DATA_BLOCK "INST_GN BLOKADA_SRUBY_LEWY"
{ S7_Optimized_Access := 'TRUE' }
VERSION : 0.1
NON_RETAIN
"3STATE_PISTON_with_brake"

BEGIN

END_DATA_BLOCK

DATA_BLOCK "INST_GN BLOKADA_SRUBY_SRODEK"
{ S7_Optimized_Access := 'TRUE' }
VERSION : 0.1
NON_RETAIN
"3STATE_PISTON_with_brake"

BEGIN

END_DATA_BLOCK

DATA_BLOCK "INST_GN BLOKADA_SRUBY_PRAWY"
{ S7_Optimized_Access := 'TRUE' }
VERSION : 0.1
NON_RETAIN
"3STATE_PISTON_with_brake"

BEGIN

END_DATA_BLOCK

DATA_BLOCK "INST_GN ZASUWKA"
{ S7_Optimized_Access := 'TRUE' }
VERSION : 0.1
NON_RETAIN
"3STATE_PISTON_with_brake"

BEGIN

END_DATA_BLOCK

DATA_BLOCK "INST_BR PIN_PODNOSZENIE_01"
{ S7_Optimized_Access := 'TRUE' }
VERSION : 0.1
NON_RETAIN
"3STATE_PISTON_with_brake"

BEGIN

END_DATA_BLOCK

DATA_BLOCK "INST_BR PIN_01"
{ S7_Optimized_Access := 'TRUE' }
VERSION : 0.1
NON_RETAIN
"3STATE_PISTON_with_brake"

BEGIN

END_DATA_BLOCK

DATA_BLOCK "INST_BR PIN_PODNOSZENIE_02"
{ S7_Optimized_Access := 'TRUE' }
VERSION : 0.1
NON_RETAIN
"3STATE_PISTON_with_brake"

BEGIN

END_DATA_BLOCK

DATA_BLOCK "INST_BR PIN_02"
{ S7_Optimized_Access := 'TRUE' }
VERSION : 0.1
NON_RETAIN
"3STATE_PISTON_with_brake"

BEGIN

END_DATA_BLOCK

DATA_BLOCK "INST_BR PIN_PODNOSZENIE_03"
{ S7_Optimized_Access := 'TRUE' }
VERSION : 0.1
NON_RETAIN
"3STATE_PISTON_with_brake"

BEGIN

END_DATA_BLOCK

DATA_BLOCK "INST_BR PIN_03"
{ S7_Optimized_Access := 'TRUE' }
VERSION : 0.1
NON_RETAIN
"3STATE_PISTON_with_brake"

BEGIN

END_DATA_BLOCK

DATA_BLOCK "INST_BR PIN_PODNOSZENIE_04"
{ S7_Optimized_Access := 'TRUE' }
VERSION : 0.1
NON_RETAIN
"3STATE_PISTON_with_brake"

BEGIN

END_DATA_BLOCK

DATA_BLOCK "INST_BR PIN_04"
{ S7_Optimized_Access := 'TRUE' }
VERSION : 0.1
NON_RETAIN
"3STATE_PISTON_with_brake"

BEGIN

END_DATA_BLOCK

DATA_BLOCK "INST_BR BLAT5_PRZOD"
{ S7_Optimized_Access := 'TRUE' }
VERSION : 0.1
NON_RETAIN
"3STATE_PISTON_with_brake"

BEGIN

END_DATA_BLOCK

DATA_BLOCK "INST_BR BLAT_TYL_LEWY"
{ S7_Optimized_Access := 'TRUE' }
VERSION : 0.1
NON_RETAIN
"3STATE_PISTON_with_brake"

BEGIN

END_DATA_BLOCK

DATA_BLOCK "INST_BR BLAT_TYL_PRAWY"
{ S7_Optimized_Access := 'TRUE' }
VERSION : 0.1
NON_RETAIN
"3STATE_PISTON_with_brake"

BEGIN

END_DATA_BLOCK

DATA_BLOCK "INST_ST1 PRZESUW_STACJI"
{ S7_Optimized_Access := 'TRUE' }
VERSION : 0.1
NON_RETAIN
"3STATE_PISTON_with_brake"

BEGIN

END_DATA_BLOCK

DATA_BLOCK "INST_ST1 WYSUW_MIECZA"
{ S7_Optimized_Access := 'TRUE' }
VERSION : 0.1
NON_RETAIN
"3STATE_PISTON_with_brake"

BEGIN

END_DATA_BLOCK

DATA_BLOCK "INST_ST1 MIECZ"
{ S7_Optimized_Access := 'TRUE' }
VERSION : 0.1
NON_RETAIN
"3STATE_PISTON_with_brake"

BEGIN

END_DATA_BLOCK

DATA_BLOCK "INST_ST2 PRZESUW_STACJI"
{ S7_Optimized_Access := 'TRUE' }
VERSION : 0.1
NON_RETAIN
"3STATE_PISTON_with_brake"

BEGIN

END_DATA_BLOCK

DATA_BLOCK "INST_ST2 WYSUW_MIECZA"
{ S7_Optimized_Access := 'TRUE' }
VERSION : 0.1
NON_RETAIN
"3STATE_PISTON_with_brake"

BEGIN

END_DATA_BLOCK

DATA_BLOCK "INST_ST2 MIECZ"
{ S7_Optimized_Access := 'TRUE' }
VERSION : 0.1
NON_RETAIN
"3STATE_PISTON_with_brake"

BEGIN

END_DATA_BLOCK

DATA_BLOCK "INST_ST3 MIECZ"
{ S7_Optimized_Access := 'TRUE' }
VERSION : 0.1
NON_RETAIN
"3STATE_PISTON_with_brake"

BEGIN

END_DATA_BLOCK

DATA_BLOCK "INST_ST3 ZDERZAK"
{ S7_Optimized_Access := 'TRUE' }
VERSION : 0.1
NON_RETAIN
"3STATE_PISTON_with_brake"

BEGIN

END_DATA_BLOCK

DATA_BLOCK "INST_ST3 PODNOSZENIE_MIECZA"
{ S7_Optimized_Access := 'TRUE' }
VERSION : 0.1
NON_RETAIN
"3STATE_PISTON_with_brake"

BEGIN

END_DATA_BLOCK

DATA_BLOCK "INST_ST4 MIECZ"
{ S7_Optimized_Access := 'TRUE' }
VERSION : 0.1
NON_RETAIN
"3STATE_PISTON_with_brake"

BEGIN

END_DATA_BLOCK

DATA_BLOCK "INST_ST4 ZDERZAK"
{ S7_Optimized_Access := 'TRUE' }
VERSION : 0.1
NON_RETAIN
"3STATE_PISTON_with_brake"

BEGIN

END_DATA_BLOCK

DATA_BLOCK "INST_ST4 PODNOSZENIE_MIECZA"
{ S7_Optimized_Access := 'TRUE' }
VERSION : 0.1
NON_RETAIN
"3STATE_PISTON_with_brake"

BEGIN

END_DATA_BLOCK

DATA_BLOCK "INST_ST5 PRZESUW_STACJI"
{ S7_Optimized_Access := 'TRUE' }
VERSION : 0.1
NON_RETAIN
"3STATE_PISTON_with_brake"

BEGIN

END_DATA_BLOCK

DATA_BLOCK "INST_ST5 STACJA_MALY_SKOK"
{ S7_Optimized_Access := 'TRUE' }
VERSION : 0.1
NON_RETAIN
"3STATE_PISTON_with_brake"

BEGIN

END_DATA_BLOCK

DATA_BLOCK "INST_ST5 STACJA_DUZY_SKOK"
{ S7_Optimized_Access := 'TRUE' }
VERSION : 0.1
NON_RETAIN
"3STATE_PISTON_with_brake"

BEGIN

END_DATA_BLOCK

DATA_BLOCK "INST_ST5 PIN"
{ S7_Optimized_Access := 'TRUE' }
VERSION : 0.1
NON_RETAIN
"3STATE_PISTON_with_brake"

BEGIN

END_DATA_BLOCK

DATA_BLOCK "INST_ST6 PRZESUW_STACJI"
{ S7_Optimized_Access := 'TRUE' }
VERSION : 0.1
NON_RETAIN
"3STATE_PISTON_with_brake"

BEGIN

END_DATA_BLOCK

DATA_BLOCK "INST_ST6 STACJA_MALY_SKOK"
{ S7_Optimized_Access := 'TRUE' }
VERSION : 0.1
NON_RETAIN
"3STATE_PISTON_with_brake"

BEGIN

END_DATA_BLOCK

DATA_BLOCK "INST_ST6 STACJA_DUZY_SKOK"
{ S7_Optimized_Access := 'TRUE' }
VERSION : 0.1
NON_RETAIN
"3STATE_PISTON_with_brake"

BEGIN

END_DATA_BLOCK

DATA_BLOCK "INST_ST6 PIN"
{ S7_Optimized_Access := 'TRUE' }
VERSION : 0.1
NON_RETAIN
"3STATE_PISTON_with_brake"

BEGIN

END_DATA_BLOCK

DATA_BLOCK "INST_ST7 PRZESUW_MIECZA_1L"
{ S7_Optimized_Access := 'TRUE' }
VERSION : 0.1
NON_RETAIN
"3STATE_PISTON_with_brake"

BEGIN

END_DATA_BLOCK

DATA_BLOCK "INST_ST7 PRZESUW_MIECZA_1P"
{ S7_Optimized_Access := 'TRUE' }
VERSION : 0.1
NON_RETAIN
"3STATE_PISTON_with_brake"

BEGIN

END_DATA_BLOCK

DATA_BLOCK "INST_ST7 PRZESUW_DOCISKOW"
{ S7_Optimized_Access := 'TRUE' }
VERSION : 0.1
NON_RETAIN
"3STATE_PISTON_with_brake"

BEGIN

END_DATA_BLOCK

DATA_BLOCK "INST_ST7 PRZESUW_MIECZA_Y_2L"
{ S7_Optimized_Access := 'TRUE' }
VERSION : 0.1
NON_RETAIN
"3STATE_PISTON_with_brake"

BEGIN

END_DATA_BLOCK

DATA_BLOCK "INST_ST7 MIECZ_2L"
{ S7_Optimized_Access := 'TRUE' }
VERSION : 0.1
NON_RETAIN
"3STATE_PISTON_with_brake"

BEGIN

END_DATA_BLOCK

DATA_BLOCK "INST_ST7 PRZESUW_MIECZA_Y_2P"
{ S7_Optimized_Access := 'TRUE' }
VERSION : 0.1
NON_RETAIN
"3STATE_PISTON_with_brake"

BEGIN

END_DATA_BLOCK

DATA_BLOCK "INST_ST7 MIECZ_2P"
{ S7_Optimized_Access := 'TRUE' }
VERSION : 0.1
NON_RETAIN
"3STATE_PISTON_with_brake"

BEGIN

END_DATA_BLOCK

DATA_BLOCK "INST_ST7 PRZESUW_MIECZA_X_3L"
{ S7_Optimized_Access := 'TRUE' }
VERSION : 0.1
NON_RETAIN
"3STATE_PISTON_with_brake"

BEGIN

END_DATA_BLOCK

DATA_BLOCK "INST_ST7 PRZESUW_MIECZA_Y_3L"
{ S7_Optimized_Access := 'TRUE' }
VERSION : 0.1
NON_RETAIN
"3STATE_PISTON_with_brake"

BEGIN

END_DATA_BLOCK

DATA_BLOCK "INST_ST7 MIECZ_3L"
{ S7_Optimized_Access := 'TRUE' }
VERSION : 0.1
NON_RETAIN
"3STATE_PISTON_with_brake"

BEGIN

END_DATA_BLOCK

DATA_BLOCK "INST_ST7 PRZESUW_MIECZA_X_3P"
{ S7_Optimized_Access := 'TRUE' }
VERSION : 0.1
NON_RETAIN
"3STATE_PISTON_with_brake"

BEGIN

END_DATA_BLOCK

DATA_BLOCK "INST_ST7 PRZESUW_MIECZA_Y_3P"
{ S7_Optimized_Access := 'TRUE' }
VERSION : 0.1
NON_RETAIN
"3STATE_PISTON_with_brake"

BEGIN

END_DATA_BLOCK

DATA_BLOCK "INST_ST7 MIECZ_3P"
{ S7_Optimized_Access := 'TRUE' }
VERSION : 0.1
NON_RETAIN
"3STATE_PISTON_with_brake"

BEGIN

END_DATA_BLOCK

DATA_BLOCK "INST_ST7 WYSUW_GRZEBIENIA"
{ S7_Optimized_Access := 'TRUE' }
VERSION : 0.1
NON_RETAIN
"3STATE_PISTON_with_brake"

BEGIN

END_DATA_BLOCK

DATA_BLOCK "INST_ST7 GRZEBIEN"
{ S7_Optimized_Access := 'TRUE' }
VERSION : 0.1
NON_RETAIN
"3STATE_PISTON_with_brake"

BEGIN

END_DATA_BLOCK

